# EPICS autosave request: softglue/softGlueApp/Db/softGlue_FPGAContent_octupole_settings.req
# shift registers
file Shift_settings.req P=$(P),H=$(H),N=1
file Shift_settings.req P=$(P),H=$(H),N=2
